// TIA Portal V20 export
// export: Created 2026-07-12T13:33:04.9480619Z, ExportSetting WithDefaults, DisplayName Totally Integrated Automation Portal, DisplayVersion V20 Update 4, DisplayName TIA Portal Openness, DisplayVersion V20 Update 4, DisplayName TIA Portal Version Control Interface, DisplayVersion V20 Update 4, DisplayName STEP 7 Professional, DisplayVersion V20 Update 4, DisplayName STEP 7 Safety, DisplayVersion V20 Update 2, DisplayName WinCC Basic/Comfort/Advanced, DisplayVersion V20 Update 4, DisplayName WinCC Unified, DisplayVersion V20 Update 4
DATA_BLOCK "DB_Vission"   // DB1
{ S7_Optimized_Access := 'FALSE' }
VERSION : 0.1
// stored: AutoNumber true, IsOnlyStoredInLoadMemory false, IsWriteProtectedInAS false
   VAR RETAIN
      bTrigger : Bool;
      iBoardWidth : Int;
      bAck : Bool;
      bResultValid : Bool;
      bError : Bool;
      wSawWord : Word;
      iLengthMM : Int;
      iWidthMM : Int;
      iBoardCount : Int;
      iErrorCode : Int;
      iHeartbeat : Int;
      iFeedSpeedCmd : Int;
      wCompareWord : Int;
      bSawDownCompare : Bool;
   END_VAR
BEGIN
END_DATA_BLOCK
